# EPICS substitutions: db/Beckhoff_3XXX/ecmcELM3604.substitutions
file "ecmcEcSlave.template"
{
  pattern {}
          {}
}

file "ecmcELM3604-chX.template"
{
  pattern {CH_ID, DTYP,             FTVL }
          {1,     asynInt32ArrayIn, LONG }
          {2,     asynInt32ArrayIn, LONG }
          {3,     asynInt32ArrayIn, LONG }
          {4,     asynInt32ArrayIn, LONG }
}
